(* IEC 61131-3 sources: verifaps-lib/stvs/src/test/resources/edu/kit/iti/formal/stvs/model/code, 3 files *)

(* ---- define_type.st ---- *)
TYPE
    MY_ENUM : (possible, values, enum);
END_TYPE

PROGRAM my_sth
    VAR_INPUT
        active : BOOL;
        number : INT;
        my_enum : MY_ENUM;
    END_VAR

    VAR_OUTPUT
        my_output : MY_ENUM;
        seriously : BOOL;
    END_VAR

    VAR
        my_enum_local : MY_ENUM;
    END_VAR

    VAR_IN_OUT
        active_inout : BOOL;
    END_VAR

END_PROGRAM

(* ---- invalidCode.st ---- *)
TYPE
     enumD : (literalOne, literalTwo);
END_TYPE

PROGRAM constantprogram
    VAR_INPUT
        A : INT;
        B : BOOL;
    END_VAR

    VAR_OUTPUT
        C : INT;
        D : enumD;
    END_VAR

    C := 52;
    öekjfdhaskljfh
END_PROGRAM

(* ---- simpleCorrectCode.st ---- *)
TYPE
  enumD : (literalOne, literalTwo);
END_TYPE

PROGRAM constantprogram
  VAR_INPUT
    A : INT;
    B : BOOL;
  END_VAR
END_PROGRAM
